Omron CX-Programmer project NewProject (CX-Programmer 9.61)

# PLC NewPLC1: CP1E N30

## Global symbols (name address type ; comment)
0.00 BOOL  ; S1
0.01 BOOL  ; LS1
0.02 BOOL  ; LS2
100.00 BOOL  ; L1

## Program NewProgram1 (cyclic task 0)

### Section Section1

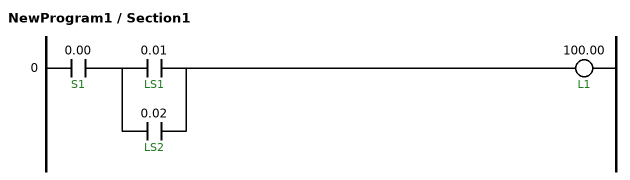
; rung 0
LD 0.00  ; S1
LD 0.01  ; LS1
OR 0.02  ; LS2
ANDLD
OUT 100.00  ; L1

### Section END
; rung 0
END(001)